TYPE ST_GOODREADPERCENTAGEOUT :
STRUCT
	GOODREADPERCENTAGECS	:STRING;
END_STRUCT
END_TYPE

(* stored: Version 1.1.0.1, ProductVersion 3.1.4024.13
   DUT ST_GOODREADPERCENTAGEOUT: Id {792ef5ad-ac84-435f-98e4-97d1fd6b380e} *)
